FUNCTION_BLOCK FbResetSet
VAR_INPUT
	xSet: BOOL;
	xReset: BOOL;
END_VAR
VAR_OUTPUT
	/// Memory 
	xQ: BOOL;
END_VAR

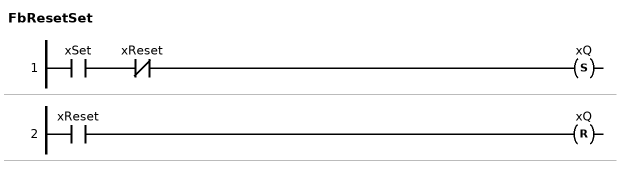
// NETWORK 1
xQ S= xSet AND NOT xReset;

// NETWORK 2
xQ R= xReset;

END_FUNCTION_BLOCK

(* stored: Version 1.1.0.1, ProductVersion 3.1.4024.12
   POU FbResetSet: Id {0447ea1c-c07c-41e9-8c2c-aba66412283e}, SpecialFunc None *)
